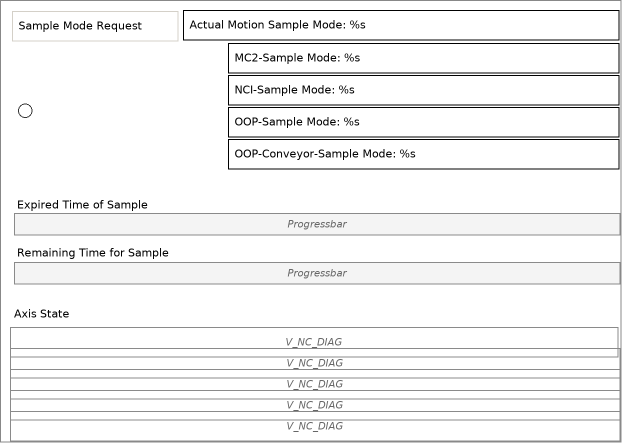
VISUALIZATION V_MAIN  // 622x443
    Rectangle (183,10 436x30), "Actual Motion Sample Mode: %s", text variable: MAIN.eSampleMode
    Rectangle (228,43 391x30), "MC2-Sample Mode: %s", text variable: MAIN.eSampleModeMC2, colour toggle: MAIN.eSampleMode = eSMode_MC2_Req
    Rectangle (228,75 391x30), "NCI-Sample Mode: %s", text variable: MAIN.eSampleModeNCI, colour toggle: MAIN.eSampleMode = eSMode_NCI_Req
    RadioButton (16,46 131x129), variable: MAIN.nRadioButton
        Areas[0]: Text=Idle
        Areas[4]: Text=OOP Convyor
    Textfield (12,11 166x30), "Sample Mode Request"
    Rectangle (228,107 391x30), "OOP-Sample Mode: %s", text variable: MAIN.eSampleModeOOP, colour toggle: MAIN.eSampleMode = eSMode_OOP_Req
    Rectangle (228,139 391x30), "OOP-Conveyor-Sample Mode: %s", text variable: MAIN.eSampleModeOOPConv, colour toggle: MAIN.eSampleMode = eSMode_OOPConv_Req
    Frame (10,327 608x30)
        shows V_NC_DIAG(AxisRef := MAIN.AxisRef[1])
    Frame (10,348 610x30)
        shows V_NC_DIAG(AxisRef := MAIN.AxisRef[2])
    Frame (10,369 610x30)
        shows V_NC_DIAG(AxisRef := MAIN.AxisRef[3])
    Frame (10,390 610x30)
        shows V_NC_DIAG(AxisRef := MAIN.AxisRef[4])
    Frame (10,411 610x30)
        shows V_NC_DIAG(AxisRef := MAIN.AxisRef[5])
    Progressbar (14,213 606x22), variable: 60-MAIN.nRemainingModeTime
    Progressbar (14,262 606x22), variable: MAIN.nRemainingModeTime
    Label (11,299 150x30), "Axis State"
    Label (14,190 150x30), "Expired Time of Sample"
    Label (14,238 225x30), "Remaining Time for Sample"
END_VISUALIZATION

(* stored: Version 1.1.0.1, ProductVersion 3.1.4024.11
   Visu V_MAIN: Id {841b37fa-a537-41e4-842b-3604596c1172} *)
